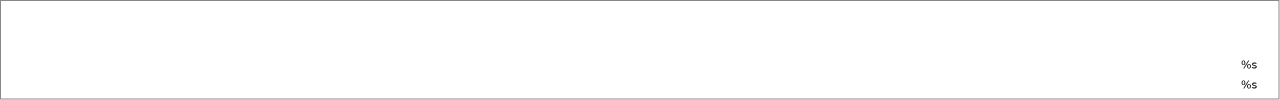
VISUALIZATION Footer_Main  // 1280x100
    Textfield (1160,70 100x30), "%s", text variable: MAIN.fb_TimeStamp.SystemDate
    Textfield (1160,50 100x30), "%s", text variable: MAIN.fb_TimeStamp.SystemTime
END_VISUALIZATION

(* stored: Version 1.1.0.1, ProductVersion 3.1.4024.12
   Visu Footer_Main: Id {1e6c3ce1-160b-4b62-b4a1-ac40fdfd577a} *)
